# EPICS autosave request: iocBoot/ioc13bmd_DAC_XPS/auto_settings.req
file "CARS_motor_settings.req",         P=$(P), M=m89
file "CARS_motor_settings.req",         P=$(P), M=m90
file "CARS_motor_settings.req",         P=$(P), M=m91
file "CARS_motor_settings.req",         P=$(P), M=m92
file "CARS_motor_settings.req",         P=$(P), M=m93
file "CARS_motor_settings.req",         P=$(P), M=m94
